PROGRAM caseTest
VAR
	motorStatus : EmotorStatus;
	shiftVal : INT := 0;
END_VAR

CASE shiftVal OF
	0: motorStatus := EmotorStatus.stopped;
	1: motorStatus := EmotorStatus.start;
	2: motorStatus := EmotorStatus.running;
END_CASE

END_PROGRAM

(* stored: Version 1.1.0.1, ProductVersion 3.1.4024.12
   POU caseTest: Id {9574d148-95dc-47f4-bbfb-4520d54ffa30}, SpecialFunc None *)
